FUNCTION_BLOCK STRING_DEMUX2N (* Basic Function Block Type *)
  (* Standard: 61499-2 *)
  (* Version 0.0, 2015-11-13, 4DIAC-IDE, 4DIAC-Consortium *)
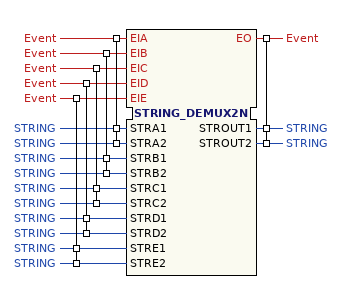
  EVENT_INPUT
    EIA WITH STRA1, STRA2;
    EIB WITH STRB1, STRB2;
    EIC WITH STRC1, STRC2;
    EID WITH STRD1, STRD2;
    EIE WITH STRE1, STRE2;
  END_EVENT
  EVENT_OUTPUT
    EO WITH STROUT1, STROUT2;
  END_EVENT
  VAR_INPUT
    STRA1 : STRING;
    STRA2 : STRING;
    STRB1 : STRING;
    STRB2 : STRING;
    STRC1 : STRING;
    STRC2 : STRING;
    STRD1 : STRING;
    STRD2 : STRING;
    STRE1 : STRING;
    STRE2 : STRING;
  END_VAR
  VAR_OUTPUT
    STROUT1 : STRING;
    STROUT2 : STRING;
  END_VAR
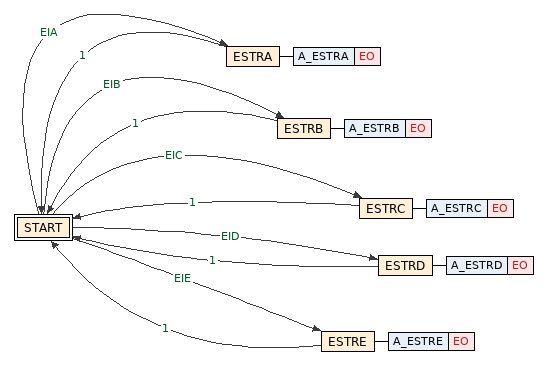
  EC_STATES
    START; (* Initial State *)
    ESTRA : A_ESTRA -> EO;
    ESTRB : A_ESTRB -> EO;
    ESTRC : A_ESTRC -> EO;
    ESTRD : A_ESTRD -> EO;
    ESTRE : A_ESTRE -> EO;
  END_STATES
  EC_TRANSITIONS
    START TO ESTRA := EIA;
    ESTRA TO START := 1;
    START TO ESTRB := EIB;
    ESTRB TO START := 1;
    START TO ESTRC := EIC;
    ESTRC TO START := 1;
    START TO ESTRD := EID;
    ESTRD TO START := 1;
    START TO ESTRE := EIE;
    ESTRE TO START := 1;
  END_TRANSITIONS
  ALGORITHM A_ESTRA IN ST: (* Initialization algorithm *)
STROUT1:=STRA1;
STROUT2:=STRA2;
  END_ALGORITHM
  ALGORITHM A_ESTRB IN ST: (* Normally executed algorithm *)
STROUT1:=STRB1;
STROUT2:=STRB2;
  END_ALGORITHM
  ALGORITHM A_ESTRC IN ST: (* new algorithm *)
STROUT1:=STRC1;
STROUT2:=STRC2;
  END_ALGORITHM
  ALGORITHM A_ESTRD IN ST: (* new algorithm *)
STROUT1:=STRD1;
STROUT2:=STRD2;
  END_ALGORITHM
  ALGORITHM A_ESTRE IN ST: (* new algorithm *)
STROUT1:=STRE1;
STROUT2:=STRE2;
  END_ALGORITHM
END_FUNCTION_BLOCK
